(* Logix 5000 project; controller Project_Template vendor 1 type 14 code 106 rev 33.12; software revision 33.00 *)

TASK MainTask (continuous, watchdog 500 ms) : MainProgram

MODULES
   Local : vendor 1 type 14 code 106 (Compact 0, rev 33.12)
      Discrete_In_Slot_3 : 1769-IQ16 (Compact 3, rev 1.1, Input RPI 20 ms)
      Discrete_In_Slot_2 : 1769-IQ16 (Compact 2, rev 1.1, Input RPI 20 ms)
      Discrete_Out_Slot_5 : 1769-OW16 (Compact 5, rev 1.1, Output RPI 20 ms)
      Discrete_Out_Slot_4 : 1769-OW16 (Compact 4, rev 1.1, Output RPI 20 ms)
      ASCII_Slot_1 : vendor 1 type 109 code 66 (Compact 1, rev 2.1, Output RPI 100 ms)
END_MODULES

VAR_GLOBAL   (* controller tags *)
   Fast_Flash_Off : TIMER := (PRE := 250, ACC := 132, EN := 1, TT := 1);
   Fast_Flash_On : TIMER := (PRE := 250, ACC := 250, EN := 1, DN := 1);
   Fast_Flasher : BOOL := 1;
   Flasher : TIMER;
   I : BOOL := 1;
   I_Auto_Mode_Selector : ALIAS FOR Local:2:I.Data.2;
   I_Barcode_Stop_Raised : ALIAS FOR Local:3:I.Data.1;
   I_Box_Ejector_Extended : ALIAS FOR Local:2:I.Data.4;
   I_Conveyor_Prox_Sensor : ALIAS FOR Local:3:I.Data.7;
   I_Reject_Cyl_Lowered : ALIAS FOR Local:3:I.Data.2;
   I_Reset_PB : ALIAS FOR Local:2:I.Data.3;
   I_Start_PB : ALIAS FOR Local:2:I.Data.0;
   I_Stop_PB : ALIAS FOR Local:2:I.Data.1;
   I_Vacuum_Head_at_Conveyor : ALIAS FOR Local:3:I.Data.0;
   I_Vacuum_Head_at_Magazine : ALIAS FOR Local:2:I.Data.15;
   I_Vacuum_Head_Extended : ALIAS FOR Local:2:I.Data.14;
   I_Vacuum_Head_Lowered : ALIAS FOR Local:2:I.Data.10;
   I_Vacuum_Head_Raised : ALIAS FOR Local:2:I.Data.9;
   I_Vacuum_Head_Retracted : ALIAS FOR Local:2:I.Data.13;
   I_Vacuum_Head_Rotated_CCW : ALIAS FOR Local:2:I.Data.11;
   I_Vacuum_Head_Rotated_CW : ALIAS FOR Local:2:I.Data.12;
   I_Vacuum_Sensor_On : ALIAS FOR Local:3:I.Data.8;
   Normal_Flash_Off : TIMER := (PRE := 500, ACC := 382, EN := 1, TT := 1);
   Normal_Flash_On : TIMER := (PRE := 500, ACC := 500, EN := 1, DN := 1);
   Normal_Flasher : BOOL := 1;
   O_Amber_Tower_Ind : ALIAS FOR Local:5:O.Data.9;
   O_Barcode_Stop_Raise : ALIAS FOR Local:4:O.Data.14;
   O_Box_Eject : ALIAS FOR Local:4:O.Data.0;
   O_Conveyor_On : ALIAS FOR Local:5:O.Data.5;
   O_Green_Tower_Ind : ALIAS FOR Local:5:O.Data.8;
   O_Red_Tower_Ind : ALIAS FOR Local:5:O.Data.10;
   O_Reject_Cyl_Extend : ALIAS FOR Local:5:O.Data.0;
   O_Reject_Cyl_Lower : ALIAS FOR Local:4:O.Data.15;
   O_Vacuum_Head_Extend : ALIAS FOR Local:4:O.Data.8;
   O_Vacuum_Head_Lower : ALIAS FOR Local:4:O.Data.5;
   O_Vacuum_Head_Rotate_CCW : ALIAS FOR Local:4:O.Data.7;
   O_Vacuum_Head_Rotate_CW : ALIAS FOR Local:4:O.Data.6;
   O_Vacuum_Head_to_Conveyor : ALIAS FOR Local:4:O.Data.9;
   O_Vacuum_Head_to_Magazine : ALIAS FOR Local:4:O.Data.10;
   O_Vacuum_Off : ALIAS FOR Local:5:O.Data.2;
   O_Vacuum_On : ALIAS FOR Local:5:O.Data.1;
   Resetting : BOOL;
   Slow_Flash_Off : TIMER := (PRE := 1000, ACC := 883, EN := 1, TT := 1);
   Slow_Flash_On : TIMER := (PRE := 1000, ACC := 1000, EN := 1, DN := 1);
   Slow_Flasher : BOOL := 1;
   Timer : TIMER[10] := ([0].PRE := 1400, [0].ACC := 38, [0].EN := 1, [0].TT := 1);
END_VAR

PROGRAM MainProgram   (* main routine MainRoutine *)
VAR
   Home : BOOL := 1;
   Production_Run : BOOL;
   Production_Running : BOOL;
   Production_Step : DINT;
   Sequence1 : BOOL;
END_VAR

ROUTINE a_Reset_Routine   (* ladder *)
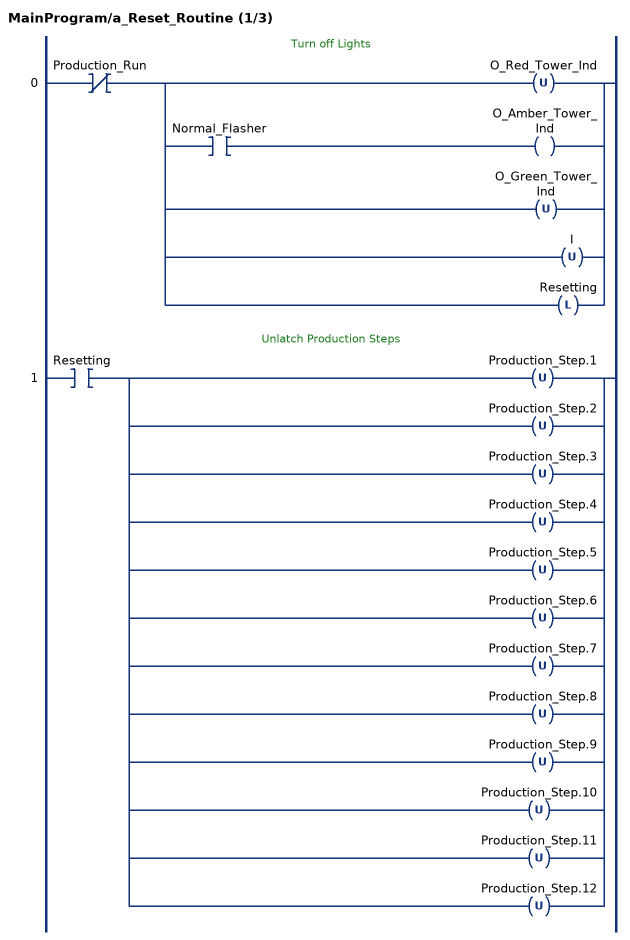
   // Turn off Lights
   0: XIO(Production_Run)[OTU(O_Red_Tower_Ind) ,XIC(Normal_Flasher) OTE(O_Amber_Tower_Ind) ,OTU(O_Green_Tower_Ind) ,OTU(I) ,OTL(Resetting) ];
   // Unlatch Production Steps
   1: XIC(Resetting)[OTU(Production_Step.1) ,OTU(Production_Step.2) ,OTU(Production_Step.3) ,OTU(Production_Step.4) ,OTU(Production_Step.5) ,OTU(Production_Step.6) ,OTU(Production_Step.7) ,OTU(Production_Step.8) ,OTU(Production_Step.9) ,OTU(Production_Step.10) ,OTU(Production_Step.11) ,OTU(Production_Step.12) ];
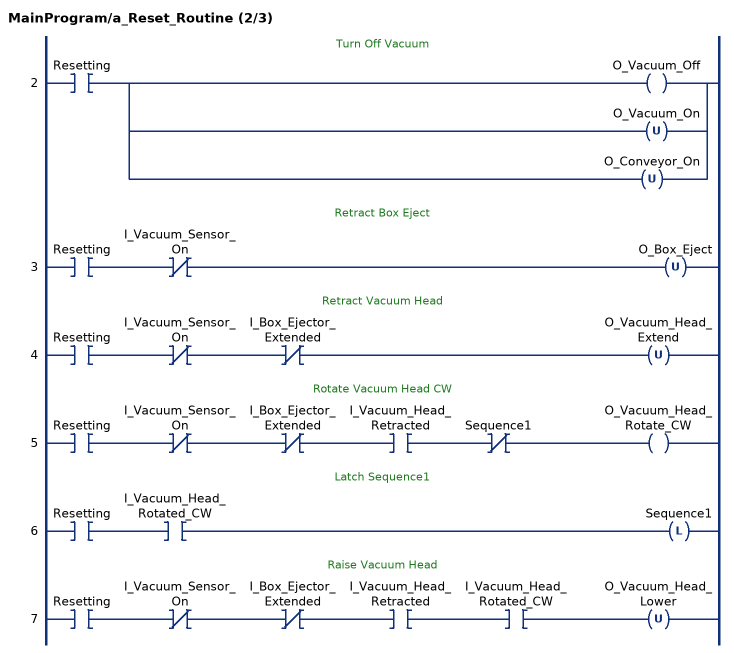
   // Turn Off Vacuum
   2: XIC(Resetting)[OTE(O_Vacuum_Off) ,OTU(O_Vacuum_On) ,OTU(O_Conveyor_On) ];
   // Retract Box Eject
   3: XIC(Resetting)XIO(I_Vacuum_Sensor_On)OTU(O_Box_Eject);
   // Retract Vacuum Head
   4: XIC(Resetting)XIO(I_Vacuum_Sensor_On)XIO(I_Box_Ejector_Extended)OTU(O_Vacuum_Head_Extend);
   // Rotate Vacuum Head CW
   5: XIC(Resetting)XIO(I_Vacuum_Sensor_On)XIO(I_Box_Ejector_Extended)XIC(I_Vacuum_Head_Retracted)XIO(Sequence1)OTE(O_Vacuum_Head_Rotate_CW);
   // Latch Sequence1
   6: XIC(Resetting)XIC(I_Vacuum_Head_Rotated_CW)OTL(Sequence1);
   // Raise Vacuum Head
   7: XIC(Resetting)XIO(I_Vacuum_Sensor_On)XIO(I_Box_Ejector_Extended)XIC(I_Vacuum_Head_Retracted)XIC(I_Vacuum_Head_Rotated_CW)OTU(O_Vacuum_Head_Lower);
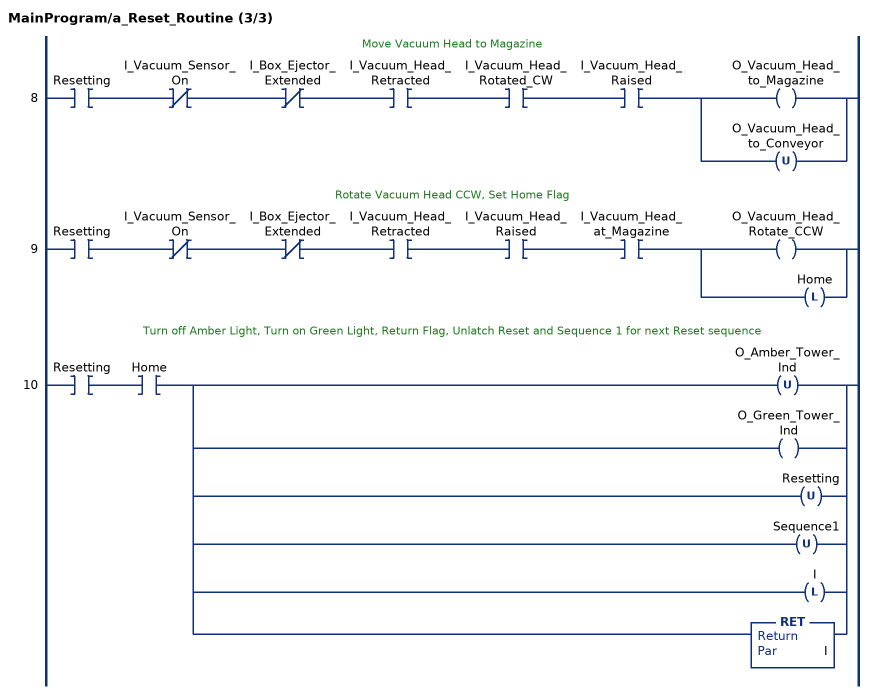
   // Move Vacuum Head to Magazine
   8: XIC(Resetting)XIO(I_Vacuum_Sensor_On)XIO(I_Box_Ejector_Extended)XIC(I_Vacuum_Head_Retracted)XIC(I_Vacuum_Head_Rotated_CW)XIC(I_Vacuum_Head_Raised)[OTE(O_Vacuum_Head_to_Magazine) ,OTU(O_Vacuum_Head_to_Conveyor) ];
   // Rotate Vacuum Head CCW, Set Home Flag
   9: XIC(Resetting)XIO(I_Vacuum_Sensor_On)XIO(I_Box_Ejector_Extended)XIC(I_Vacuum_Head_Retracted)XIC(I_Vacuum_Head_Raised)XIC(I_Vacuum_Head_at_Magazine)[OTE(O_Vacuum_Head_Rotate_CCW) ,OTL(Home) ];
   // Turn off Amber Light, Turn on Green Light, Return Flag, Unlatch Reset and Sequence 1 for next Reset sequence
   10: XIC(Resetting)XIC(Home)[OTU(O_Amber_Tower_Ind) ,OTE(O_Green_Tower_Ind) ,OTU(Resetting) ,OTU(Sequence1) ,OTL(I) ,RET(I) ];
END_ROUTINE

ROUTINE b_Production_Routine   (* ladder *)
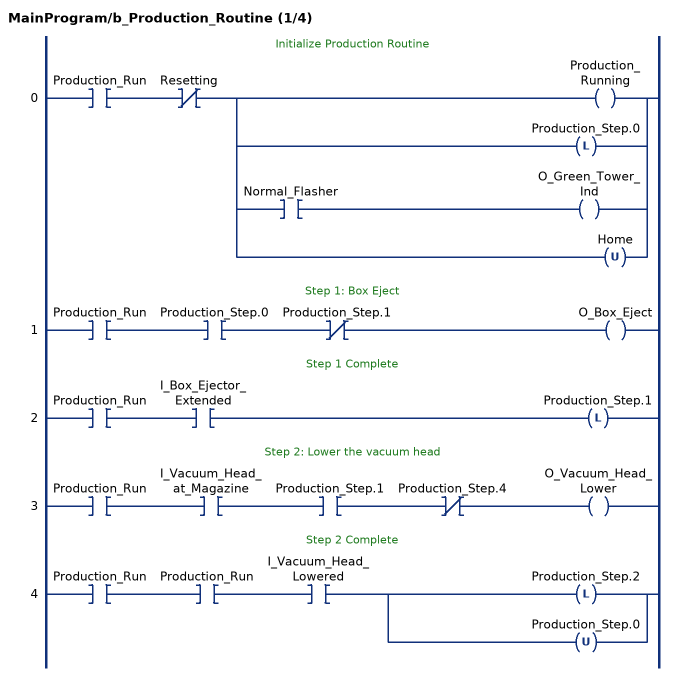
   // Initialize Production Routine
   0: XIC(Production_Run)XIO(Resetting)[OTE(Production_Running) ,OTL(Production_Step.0) ,XIC(Normal_Flasher) OTE(O_Green_Tower_Ind) ,OTU(Home) ];
   // Step 1: Box Eject
   1: XIC(Production_Run)XIC(Production_Step.0)XIO(Production_Step.1)OTE(O_Box_Eject);
   // Step 1 Complete
   2: XIC(Production_Run)XIC(I_Box_Ejector_Extended)OTL(Production_Step.1);
   // Step 2: Lower the vacuum head
   3: XIC(Production_Run)XIC(I_Vacuum_Head_at_Magazine)XIC(Production_Step.1)XIO(Production_Step.4)OTE(O_Vacuum_Head_Lower);
   // Step 2 Complete
   4: XIC(Production_Run)XIC(Production_Run)XIC(I_Vacuum_Head_Lowered)[OTL(Production_Step.2) ,OTU(Production_Step.0) ];
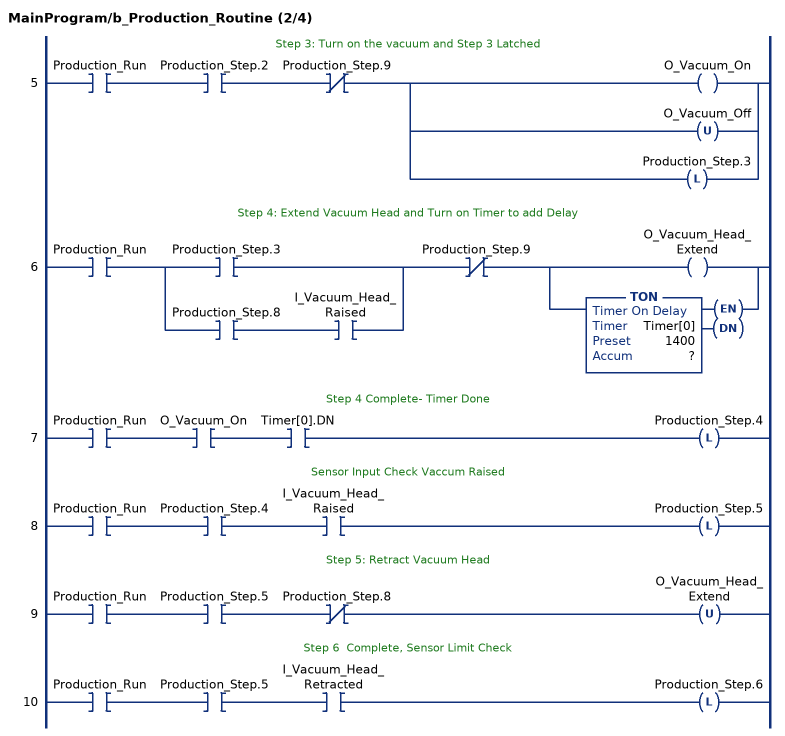
   // Step 3: Turn on the vacuum and Step 3 Latched
   5: XIC(Production_Run)XIC(Production_Step.2)XIO(Production_Step.9)[OTE(O_Vacuum_On) ,OTU(O_Vacuum_Off) ,OTL(Production_Step.3) ];
   // Step 4: Extend Vacuum Head and Turn on Timer to add Delay
   6: XIC(Production_Run)[XIC(Production_Step.3) ,XIC(Production_Step.8) XIC(I_Vacuum_Head_Raised) ]XIO(Production_Step.9)[OTE(O_Vacuum_Head_Extend) ,TON(Timer[0],?,?) ];
   // Step 4 Complete- Timer Done
   7: XIC(Production_Run)XIC(O_Vacuum_On)XIC(Timer[0].DN)OTL(Production_Step.4);
   // Sensor Input Check Vaccum Raised
   8: XIC(Production_Run)XIC(Production_Step.4)XIC(I_Vacuum_Head_Raised)OTL(Production_Step.5);
   // Step 5: Retract Vacuum Head
   9: XIC(Production_Run)XIC(Production_Step.5)XIO(Production_Step.8)OTU(O_Vacuum_Head_Extend);
   // Step 6  Complete, Sensor Limit Check
   10: XIC(Production_Run)XIC(Production_Step.5)XIC(I_Vacuum_Head_Retracted)OTL(Production_Step.6);
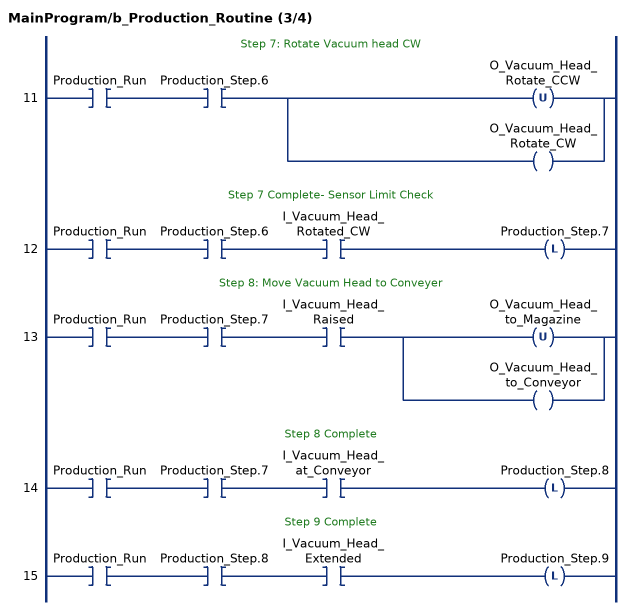
   // Step 7: Rotate Vacuum head CW
   11: XIC(Production_Run)XIC(Production_Step.6)[OTU(O_Vacuum_Head_Rotate_CCW) ,OTE(O_Vacuum_Head_Rotate_CW) ];
   // Step 7 Complete- Sensor Limit Check
   12: XIC(Production_Run)XIC(Production_Step.6)XIC(I_Vacuum_Head_Rotated_CW)OTL(Production_Step.7);
   // Step 8: Move Vacuum Head to Conveyer
   13: XIC(Production_Run)XIC(Production_Step.7)XIC(I_Vacuum_Head_Raised)[OTU(O_Vacuum_Head_to_Magazine) ,OTE(O_Vacuum_Head_to_Conveyor) ];
   // Step 8 Complete
   14: XIC(Production_Run)XIC(Production_Step.7)XIC(I_Vacuum_Head_at_Conveyor)OTL(Production_Step.8);
   // Step 9 Complete
   15: XIC(Production_Run)XIC(Production_Step.8)XIC(I_Vacuum_Head_Extended)OTL(Production_Step.9);
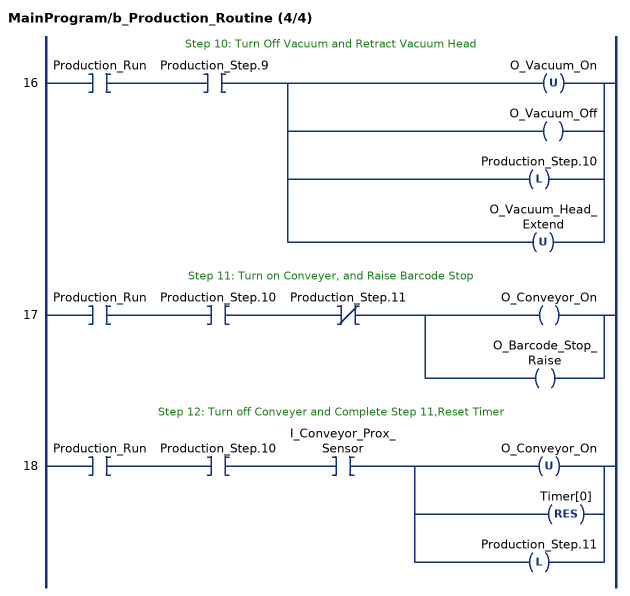
   // Step 10: Turn Off Vacuum and Retract Vacuum Head
   16: XIC(Production_Run)XIC(Production_Step.9)[OTU(O_Vacuum_On) ,OTE(O_Vacuum_Off) ,OTL(Production_Step.10) ,OTU(O_Vacuum_Head_Extend) ];
   // Step 11: Turn on Conveyer, and Raise Barcode Stop
   17: XIC(Production_Run)XIC(Production_Step.10)XIO(Production_Step.11)[OTE(O_Conveyor_On) ,OTE(O_Barcode_Stop_Raise) ];
   // Step 12: Turn off Conveyer and Complete Step 11,Reset Timer
   18: XIC(Production_Run)XIC(Production_Step.10)XIC(I_Conveyor_Prox_Sensor)[OTU(O_Conveyor_On) ,RES(Timer[0]) ,OTL(Production_Step.11) ];
END_ROUTINE

ROUTINE MainRoutine   (* ladder *)
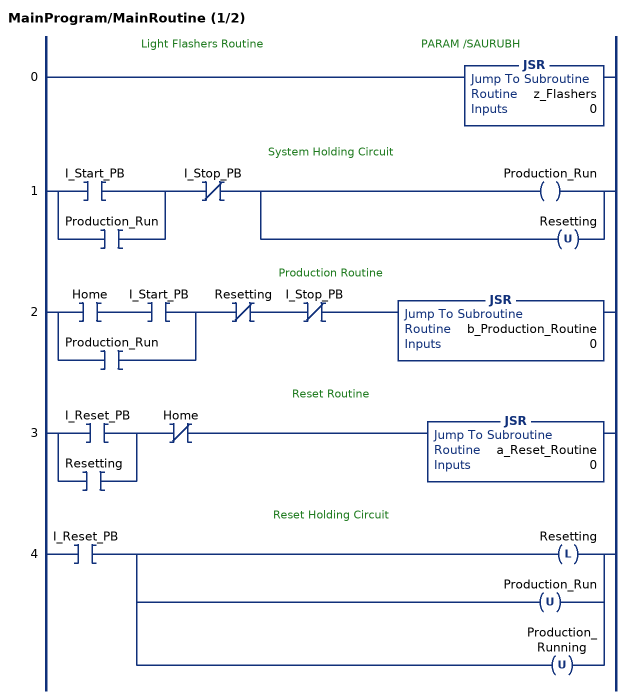
   // Light Flashers Routine                                             PARAM /SAURUBH
   0: JSR(z_Flashers,0);
   // System Holding Circuit
   1: [XIC(I_Start_PB) ,XIC(Production_Run) ]XIO(I_Stop_PB)[OTE(Production_Run) ,OTU(Resetting) ];
   // Production Routine
   2: [XIC(Home) XIC(I_Start_PB) ,XIC(Production_Run) ]XIO(Resetting)XIO(I_Stop_PB)JSR(b_Production_Routine,0);
   // Reset Routine
   3: [XIC(I_Reset_PB) ,XIC(Resetting) ]XIO(Home)JSR(a_Reset_Routine,0);
   // Reset Holding Circuit
   4: XIC(I_Reset_PB)[OTL(Resetting) ,OTU(Production_Run) ,OTU(Production_Running) ];
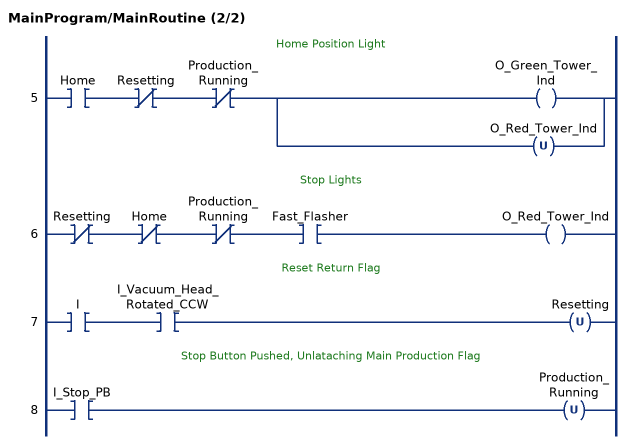
   // Home Position Light
   5: XIC(Home)XIO(Resetting)XIO(Production_Running)[OTE(O_Green_Tower_Ind) ,OTU(O_Red_Tower_Ind) ];
   // Stop Lights
   6: XIO(Resetting)XIO(Home)XIO(Production_Running)XIC(Fast_Flasher)OTE(O_Red_Tower_Ind);
   // Reset Return Flag
   7: XIC(I)XIC(I_Vacuum_Head_Rotated_CCW)OTU(Resetting);
   // Stop Button Pushed, Unlataching Main Production Flag
   8: XIC(I_Stop_PB)OTU(Production_Running);
END_ROUTINE

ROUTINE z_Flashers   (* ladder *)
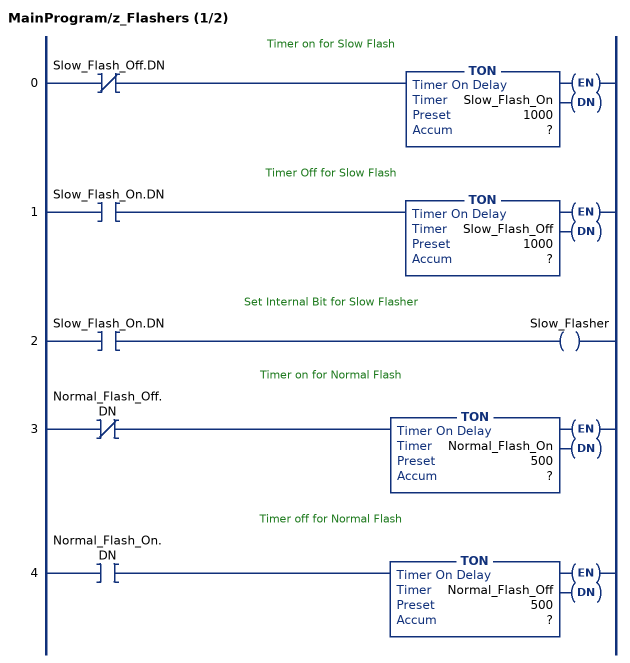
   // Timer on for Slow Flash
   0: XIO(Slow_Flash_Off.DN)TON(Slow_Flash_On,?,?);
   // Timer Off for Slow Flash
   1: XIC(Slow_Flash_On.DN)TON(Slow_Flash_Off,?,?);
   // Set Internal Bit for Slow Flasher
   2: XIC(Slow_Flash_On.DN)OTE(Slow_Flasher);
   // Timer on for Normal Flash
   3: XIO(Normal_Flash_Off.DN)TON(Normal_Flash_On,?,?);
   // Timer off for Normal Flash
   4: XIC(Normal_Flash_On.DN)TON(Normal_Flash_Off,?,?);
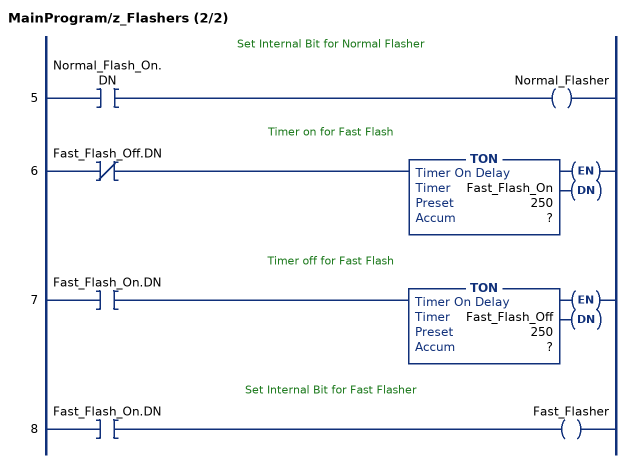
   // Set Internal Bit for Normal Flasher
   5: XIC(Normal_Flash_On.DN)OTE(Normal_Flasher);
   // Timer on for Fast Flash
   6: XIO(Fast_Flash_Off.DN)TON(Fast_Flash_On,?,?);
   // Timer off for Fast Flash
   7: XIC(Fast_Flash_On.DN)TON(Fast_Flash_Off,?,?);
   // Set Internal Bit for Fast Flasher
   8: XIC(Fast_Flash_On.DN)OTE(Fast_Flasher);
END_ROUTINE
END_PROGRAM
